// TIA Portal project "0000" (V15.1)

(* hardware
DEVICE "S7-1200-Station_1"  S7-1200 Station
   slot 0: "Baugruppenträger_0"  S7-1200 Rack  Rack  V1.0
   slot 1: "0000"  CPU 1214C DC/DC/DC  6ES7 214-1AG40-0XB0  V4.3
DEVICE "S7300/ET200M-Station_1"  S7-300 station
   slot 0: "Profilschiene_0"  Rail  6ES7 390-1***0-0AA0
   slot 2: "0001"  CPU 317-2 PN/DP  6ES7 317-2EK13-0AB0  V2.6
      slot 1: "MPI/DP-Schnittstelle_1"  X1
      slot 2: "PROFINET-Schnittstelle_1"  PN-IO
         slot 1: "Port_1"  Port
*)

// ===== PLC "0000"  CPU 1214C DC/DC/DC =====

VAR_GLOBAL   // PLC tag table "Standard-Variablentabelle"
   "Clock_Byte" AT %MB1 : Byte;
   "Clock_10Hz" AT %M1.0 : Bool;
   "Clock_5Hz" AT %M1.1 : Bool;
   "Clock_2.5Hz" AT %M1.2 : Bool;
   "Clock_2Hz" AT %M1.3 : Bool;
   "Clock_1.25Hz" AT %M1.4 : Bool;
   "Clock_1Hz" AT %M1.5 : Bool;
   "Clock_0.625Hz" AT %M1.6 : Bool;
   "Clock_0.5Hz" AT %M1.7 : Bool;
   "System_Byte" AT %MB0 : Byte;
   "FirstScan" AT %M0.0 : Bool;
   "DiagStatusUpdate" AT %M0.1 : Bool;
   "AlwaysTRUE" AT %M0.2 : Bool;
   "AlwaysFALSE" AT %M0.3 : Bool;
   "Enable_Communication" AT %M100.0 : Bool;
   "Save_Data" AT %M100.1 : Bool;
END_VAR

TYPE "_CSV_Data_UDT"
   STRUCT
      "example Bool" : Bool;   // this is a comment for Bool in UDT
   END_STRUCT;
END_TYPE

TYPE "_CSV_Data"
TITLE = has no title
// some comment
   STRUCT
      Save_Data : Bool := True;   // Trigger to save the data
      example_Byte : Byte := 16#2;   // this is a comment for example_Byte
      example_Word : Word := 16#FF;   // this is a comment for this is a comment for example_Word
      example_Dword : DWord := 16#FFFF;   // this is a comment for example_Dword
      example_Int : Int := 3;   // this is a comment for example_Int
      example_Dint : DInt := 5;   // this is a comment for example_Dint
      example_String : String := 'This is an example Text';   // this is a comment for example_String
      example_array : Array[0..5] of Bool;   // this is a comment for example_array
      example_UDT : "_CSV_Data_UDT";   // this is a comment for example UDT
   END_STRUCT;
END_TYPE

DATA_BLOCK "ConPlc_DB"   // DB1
{ S7_Optimized_Access := 'TRUE' }
VERSION : 0.1
// stored: InstanceOfName ConPlc
"ConPlc"
BEGIN
END_DATA_BLOCK

DATA_BLOCK "CSV"   // DB3
{ S7_Optimized_Access := 'FALSE' }
VERSION : 0.1
   VAR
      Data : "_CSV_Data";
   END_VAR
BEGIN
END_DATA_BLOCK

FUNCTION_BLOCK "ConPlc"   // FB1000, SCL
{ S7_Optimized_Access := 'TRUE' }
VERSION : 0.1
   VAR_INPUT
      ACTIVATE : Bool := False;   // activate connection
      TACT : Bool := False;   // tact
      CONN_ID : Conn_Ouc := 16#1;   // connection reference / identifier
      HW_ID : Hw_Any := 64;   // HW-identifier of IE-interface submodule
      CONN_Type : Byte := 16#0B;   // type of connection: 11=TCP/IP, 19=UDP (17=TCP/IP)
      IP_ADDR_1 : Byte := 16#C0;   // IPv4 address
      IP_ADDR_2 : Byte := 16#A8;   // IPv4 address
      IP_ADDR_3 : Byte := 16#00;   // IPv4 address
      IP_ADDR_4 : Byte := 16#1E;   // IPv4 address
      PORT_Remote : UInt := 2000;   // remote UDP/TCP port number
      PORT_Local : UInt := 2000;   // local UDP/TCP port number
   END_VAR
   VAR_OUTPUT
      Saved : Bool := False;   // CSV is saved
      Recieved : Bool := False;   // Data is recieved
   END_VAR
   VAR_IN_OUT
      DATA : Variant;
   END_VAR
   VAR
      ACT_CONN : Bool;
      CONN_ESTABLISHED : Bool;
      DONE_CONN : Bool;
      BUSY_CONN : Bool;
      ERROR_CONN : Bool;
      STATUS_CONN : Word;
      DONE_SEND : Bool;
      BUSY_SEND : Bool;
      ERROR_SEND : Bool;
      STATUS_SEND : Word;
      ACT_SEND : Bool;
      NDR_RECV : Bool;
      BUSY_RECV : Bool;
      ERROR_RECV : Bool;
      STATUS_RECV : Word;
      RCVD_LEN : UDInt;
      ACT_RECV : Bool;
      DONE_DISCON : Bool;
      BUSY_DISCON : Bool;
      ERROR_DISCON : Bool;
      STATUS_DISCON : Word;
      ACT_DISCON : Bool;
      TRIGGER : Bool;
      TRIGGER_MEM : Bool;
      RECV : Array[0..9] of Char;
      TCON_IDB : TCON;
      TSEND_IDB : TSEND;
      TRCV_IDB : TRCV;
      TDISCON_IDB : TDISCON;
      CONN_PARAMETER : TCON_IP_v4;
      TON_RESET : TON_TIME;
   END_VAR
   VAR_TEMP
      recv_str : String[10];
   END_VAR
   // CONN_PARAMETER.InterfaceId := 64;
   // CONN_PARAMETER.ID := 16#1;
   // CONN_PARAMETER.ConnectionType := 16#0B;
   // CONN_PARAMETER.ActiveEstablished := False;
   // CONN_PARAMETER.RemoteAddress.ADDR[1] := 16#C0;
   // CONN_PARAMETER.RemoteAddress.ADDR[2] := 16#A8;
   // CONN_PARAMETER.RemoteAddress.ADDR[3] := 16#00;
   // CONN_PARAMETER.RemoteAddress.ADDR[4] := 16#1E;
   // CONN_PARAMETER.RemotePort := 2000;
   // CONN_PARAMETER.LocalPort := 2000;
BEGIN
   REGION set connection data
       #CONN_PARAMETER.ID := #CONN_ID;
       #CONN_PARAMETER.InterfaceId := #HW_ID;
       #CONN_PARAMETER.ActiveEstablished := TRUE;
       #CONN_PARAMETER.ConnectionType := #CONN_Type;
       #CONN_PARAMETER.RemoteAddress.ADDR[1] := #IP_ADDR_1;
       #CONN_PARAMETER.RemoteAddress.ADDR[2] := #IP_ADDR_2;
       #CONN_PARAMETER.RemoteAddress.ADDR[3] := #IP_ADDR_3;
       #CONN_PARAMETER.RemoteAddress.ADDR[4] := #IP_ADDR_4;
       #CONN_PARAMETER.RemotePort := #PORT_Remote;
       #CONN_PARAMETER.LocalPort := #PORT_Local;
   END_REGION

   REGION create trigger
       #TRIGGER := #TACT AND NOT #TRIGGER_MEM;
       #TRIGGER_MEM := #TACT;
   END_REGION

   REGION connect
       //connect enable
       IF #ACTIVATE AND NOT #CONN_ESTABLISHED THEN
           #ACT_CONN := True;
       END_IF;
       //connect
       #TCON_IDB(REQ       := #ACT_CONN AND #TRIGGER,
                 ID        := #CONN_ID,
                 DONE      => #DONE_CONN,
                 BUSY      => #BUSY_CONN,
                 ERROR     => #ERROR_CONN,
                 STATUS    => #STATUS_CONN,
                 CONNECT   := #CONN_PARAMETER);
       //connect done
       IF #DONE_CONN THEN
           #CONN_ESTABLISHED := True;
           #ACT_CONN := False;
       END_IF;
   END_REGION

   REGION send
       //send enable
       #ACT_SEND := #CONN_ESTABLISHED AND #TRIGGER AND NOT #BUSY_SEND;
       //send
       #TSEND_IDB(REQ      := #ACT_SEND,
                  ID       := #CONN_ID,
                  LEN      := 0,
                  DONE     => #DONE_SEND,
                  BUSY     => #BUSY_SEND,
                  ERROR    => #ERROR_SEND,
                  STATUS   => #STATUS_SEND,
                  DATA     := #DATA);
   END_REGION

   REGION recieve

       //revieve enable
       #ACT_RECV := #CONN_ESTABLISHED;
       //recieve
       #TRCV_IDB(EN_R      := #ACT_RECV,
                 ID        := #CONN_ID,
                 LEN       := 10,
                 ADHOC     := TRUE,
                 NDR       => #NDR_RECV,
                 BUSY      => #BUSY_RECV,
                 ERROR     => #ERROR_RECV,
                 STATUS    => #STATUS_RECV,
                 RCVD_LEN  => #RCVD_LEN,
                 DATA      := #RECV);

       //put recieved Bytes in String
       Chars_TO_Strg(Chars:=#RECV, pChars:=0, Cnt:=10, Strg=>#recv_str);

       //check recieved data
       #Saved := #NDR_RECV AND (#recv_str = 'Saved     ');
       #Recieved := #NDR_RECV AND (#recv_str = 'Recieved  ');

   END_REGION

   REGION disconnect
       //disconnect enable
       #TON_RESET(IN := #ACTIVATE AND NOT #CONN_ESTABLISHED,
                  PT := T#5s);
       #ACT_DISCON := (#TON_RESET.Q) OR (NOT #ACTIVATE);
       //disconnect
       #TDISCON_IDB(REQ    := #ACT_DISCON,
                    ID     := #CONN_ID,
                    DONE   => #DONE_DISCON,
                    BUSY   => #BUSY_DISCON,
                    ERROR  => #ERROR_DISCON,
                    STATUS => #STATUS_DISCON);

       //disconnect done
       IF NOT #ACTIVATE THEN
           #CONN_ESTABLISHED := False;
           #ACT_CONN := False;
       END_IF;
   END_REGION
END_FUNCTION_BLOCK

ORGANIZATION_BLOCK "Main"   // OB1, FBD, ProgramCycle
TITLE = "Main Program Sweep (Cycle)"
{ S7_Optimized_Access := 'TRUE' }
VERSION : 0.1
   VAR_INPUT
      Initial_Call : Bool;   // Initial call of this OB
      Remanence : Bool;   // =True, if remanent data are available
   END_VAR
   VAR_TEMP
      retval : Int;
      saved : Bool;
      recieved : Bool;
   END_VAR
BEGIN

REGION Network 1: Collect Data
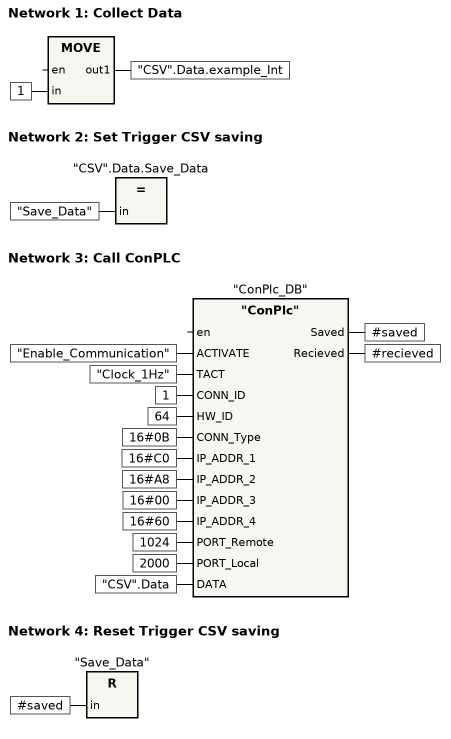
   "CSV".Data.example_Int := 1;
END_REGION

REGION Network 2: Set Trigger CSV saving
   "CSV".Data.Save_Data := "Save_Data";
END_REGION

REGION Network 3: Call ConPLC
   "ConPlc_DB"(ACTIVATE := "Enable_Communication",   // "ConPlc"
               TACT := "Clock_1Hz",
               CONN_ID := 1,
               HW_ID := 64,
               CONN_Type := 16#0B,
               IP_ADDR_1 := 16#C0,
               IP_ADDR_2 := 16#A8,
               IP_ADDR_3 := 16#00,
               IP_ADDR_4 := 16#60,
               PORT_Remote := 1024,
               PORT_Local := 2000,
               DATA := "CSV".Data,
               Saved => #saved,
               Recieved => #recieved);
END_REGION

REGION Network 4: Reset Trigger CSV saving
   IF #saved THEN "Save_Data" := FALSE; END_IF;
END_REGION
END_ORGANIZATION_BLOCK

// ===== PLC "0001"  CPU 317-2 PN/DP =====

VAR_GLOBAL   // PLC tag table "Standard-Variablentabelle"
   "Clock_Byte" AT %MB1 : Byte;
   "Clock_10Hz" AT %M1.0 : Bool;
   "Clock_5Hz" AT %M1.1 : Bool;
   "Clock_2.5Hz" AT %M1.2 : Bool;
   "Clock_2Hz" AT %M1.3 : Bool;
   "Clock_1.25Hz" AT %M1.4 : Bool;
   "Clock_1Hz" AT %M1.5 : Bool;
   "Clock_0.625Hz" AT %M1.6 : Bool;
   "Clock_0.5Hz" AT %M1.7 : Bool;
   "Enable_Communication" AT %M100.0 : Bool;
   "Save_Data" AT %M100.1 : Bool;
END_VAR

TYPE "_CSV_Data_UDT"
   STRUCT
      "example Bool" : Bool;   // this is a comment for Bool in UDT
   END_STRUCT;
END_TYPE

TYPE "_CSV_Data"
TITLE = has no title
// some comment
   STRUCT
      Save_Data : Bool := True;   // Trigger to save the data
      example_Byte : Byte := 16#2;   // this is a comment for example_Byte
      example_Word : Word := 16#FF;   // this is a comment for this is a comment for example_Word
      example_Dword : DWord := 16#FFFF;   // this is a comment for example_Dword
      example_Int : Int := 3;   // this is a comment for example_Int
      example_Dint : DInt := 5;   // this is a comment for example_Dint
      example_String : String := 'This is an example Text';   // this is a comment for example_String
      example_array : Array[0..5] of Bool;   // this is a comment for example_array
      example_UDT : "_CSV_Data_UDT";   // this is a comment for example UDT
   END_STRUCT;
END_TYPE

DATA_BLOCK "ConPlc_DB"   // DB1
{ S7_Optimized_Access := 'FALSE' }
VERSION : 0.1
// stored: InstanceOfName ConPlc
"ConPlc"
BEGIN
   ACTIVATE := TRUE;
   TACT := TRUE;
   CONN_ID := 16#0001;
   Saved := FALSE;
   Recieved := FALSE;
   DATA := P#DB3.DBX0.0 BYTE 274;
   ACT_CONN := TRUE;
   STATUS_CONN := 16#7000;
   STATUS_SEND := 16#7000;
   STATUS_RECV := 16#7000;
   STATUS_DISCON := 16#7000;
   ACT_DISCON := TRUE;
   TRIGGER := TRUE;
   TRIGGER_MEM := TRUE;
   RECV[0] := ' ';
   RECV[1] := ' ';
   RECV[2] := ' ';
   RECV[3] := ' ';
   RECV[4] := ' ';
   RECV[5] := ' ';
   RECV[6] := ' ';
   RECV[7] := ' ';
   RECV[8] := ' ';
   RECV[9] := ' ';
   TCON_IDB.REQ := TRUE;
   TCON_IDB.ID := 16#0001;
   TCON_IDB.STATUS := 16#7000;
   TCON_IDB.CONNECT := P#DB1.DBX122.0 BYTE 64;
   TSEND_IDB.ID := 16#0001;
   TSEND_IDB.STATUS := 16#7000;
   TSEND_IDB.DATA := P#DB3.DBX0.0 BYTE 274;
   TRCV_IDB.ID := 16#0001;
   TRCV_IDB.LEN := 10;
   TRCV_IDB.STATUS := 16#7000;
   TRCV_IDB.DATA := P#DB1.DBX36.0 CHAR 10;
   TDISCON_IDB.REQ := TRUE;
   TDISCON_IDB.ID := 16#0001;
   TDISCON_IDB.STATUS := 16#7000;
   TON_RESET.IN := TRUE;
   TON_RESET.PT := T#5S;
   TON_RESET.Q := TRUE;
   TON_RESET.ET := T#5S;
END_DATA_BLOCK

DATA_BLOCK "CSV"   // DB3
{ S7_Optimized_Access := 'FALSE' }
VERSION : 0.1
   VAR
      Data : "_CSV_Data";
   END_VAR
BEGIN
END_DATA_BLOCK

FUNCTION_BLOCK "ConPlc"   // FB1000, SCL
{ S7_Optimized_Access := 'FALSE' }
VERSION : 0.1
   VAR_INPUT
      ACTIVATE : Bool := False;   // activate connection
      TACT : Bool := False;   // tact
      CONN_ID : Word := 16#1;   // connection reference / identifier
   END_VAR
   VAR_OUTPUT
      Saved : Bool := False;   // CSV is saved
      Recieved : Bool := False;   // Data is recieved
   END_VAR
   VAR_IN_OUT
      DATA : ANY;
   END_VAR
   VAR
      ACT_CONN : Bool;
      CONN_ESTABLISHED : Bool;
      DONE_CONN : Bool;
      BUSY_CONN : Bool;
      ERROR_CONN : Bool;
      STATUS_CONN : Word;
      DONE_SEND : Bool;
      BUSY_SEND : Bool;
      ERROR_SEND : Bool;
      STATUS_SEND : Word;
      ACT_SEND : Bool;
      NDR_RECV : Bool;
      BUSY_RECV : Bool;
      ERROR_RECV : Bool;
      STATUS_RECV : Word;
      RCVD_LEN : Int;
      ACT_RECV : Bool;
      DONE_DISCON : Bool;
      BUSY_DISCON : Bool;
      ERROR_DISCON : Bool;
      STATUS_DISCON : Word;
      ACT_DISCON : Bool;
      TRIGGER : Bool;
      TRIGGER_MEM : Bool;
      RECV : Array[0..9] of Char;
      TCON_IDB : TCON;
      TSEND_IDB : TSEND;
      TRCV_IDB : TRCV;
      TDISCON_IDB : TDISCON;
      CONN_PARAMETER : TCON_PAR;
      TON_RESET : TON;
   END_VAR
   VAR_TEMP
      recv_str : String[10];
      cnt : Int;
      retval : Int;
   END_VAR
BEGIN
   REGION create trigger
       #TRIGGER := #TACT AND NOT #TRIGGER_MEM;
       #TRIGGER_MEM := #TACT;
   END_REGION

   REGION connect
       //connect enable
       IF #ACTIVATE AND NOT #CONN_ESTABLISHED THEN
           #ACT_CONN := True;
       END_IF;

       //connect
       #TCON_IDB(REQ       := #ACT_CONN AND #TRIGGER,
                 ID        := #CONN_ID,
                 DONE      => #DONE_CONN,
                 BUSY      => #BUSY_CONN,
                 ERROR     => #ERROR_CONN,
                 STATUS    => #STATUS_CONN,
                 CONNECT   := #CONN_PARAMETER);
       //connect done
       IF #DONE_CONN THEN
           #CONN_ESTABLISHED := True;
           #ACT_CONN := False;
       END_IF;
   END_REGION

   REGION send
       //send enable
       #ACT_SEND := #CONN_ESTABLISHED AND #TRIGGER AND NOT #BUSY_SEND;
       //send
       #TSEND_IDB(REQ      := #ACT_SEND,
                  ID       := #CONN_ID,
                  LEN      := 0,
                  DONE     => #DONE_SEND,
                  BUSY     => #BUSY_SEND,
                  ERROR    => #ERROR_SEND,
                  STATUS   => #STATUS_SEND,
                  DATA     := #DATA);
   END_REGION

   REGION recieve

       //revieve enable
       #ACT_RECV := #CONN_ESTABLISHED;
       //recieve
       #TRCV_IDB(EN_R      := #ACT_RECV,
                 ID        := #CONN_ID,
                 LEN       := 10,
                 NDR       => #NDR_RECV,
                 BUSY      => #BUSY_RECV,
                 ERROR     => #ERROR_RECV,
                 STATUS    => #STATUS_RECV,
                 RCVD_LEN  => #RCVD_LEN,
                 DATA      := #RECV);

       //put recieved Bytes in String
       #retval := BLKMOV(SRCBLK:=#RECV, DSTBLK=>#recv_str);

       //check recieved data
       #Saved := #NDR_RECV AND (#recv_str S_COMP 'Saved     ');
       #Recieved := #NDR_RECV AND (#recv_str S_COMP 'Recieved  ');

   END_REGION

   REGION disconnect
       //disconnect enable
       #TON_RESET(IN := #ACTIVATE AND NOT #CONN_ESTABLISHED,
                  PT := T#5s);
       #ACT_DISCON := (#TON_RESET.Q) OR (NOT #ACTIVATE);
       //disconnect
       #TDISCON_IDB(REQ    := #ACT_DISCON,
                    ID     := #CONN_ID,
                    DONE   => #DONE_DISCON,
                    BUSY   => #BUSY_DISCON,
                    ERROR  => #ERROR_DISCON,
                    STATUS => #STATUS_DISCON);

       //disconnect done
       IF NOT #ACTIVATE THEN
           #CONN_ESTABLISHED := False;
           #ACT_CONN := False;
       END_IF;
   END_REGION
END_FUNCTION_BLOCK

ORGANIZATION_BLOCK "Main"   // OB1, FBD
TITLE = "Main Program Sweep (Cycle)"
{ S7_Optimized_Access := 'FALSE' }
VERSION : 0.1
   VAR_TEMP
      OB1_EV_CLASS : Byte;   // Bits 0-3 = 1 (Coming event), Bits 4-7 = 1 (Event class 1)
      OB1_SCAN_1 : Byte;   // 1 (Cold restart scan 1 of OB 1), 3 (Scan 2-n of OB 1)
      OB1_PRIORITY : Byte;   // Priority of OB Execution
      OB1_OB_NUMBR : Byte;   // 1 (Organization block 1, OB1)
      OB1_RESERVED_1 : Byte;   // Reserved for system
      OB1_RESERVED_2 : Byte;   // Reserved for system
      OB1_PREV_CYCLE : Int;   // Cycle time of previous OB1 scan (milliseconds)
      OB1_MIN_CYCLE : Int;   // Minimum cycle time of OB1 (milliseconds)
      OB1_MAX_CYCLE : Int;   // Maximum cycle time of OB1 (milliseconds)
      OB1_DATE_TIME : Date_And_Time;   // Date and time OB1 started
      saved : Bool;
      recieved : Bool;
   END_VAR
BEGIN

REGION Network 1: Collect Data
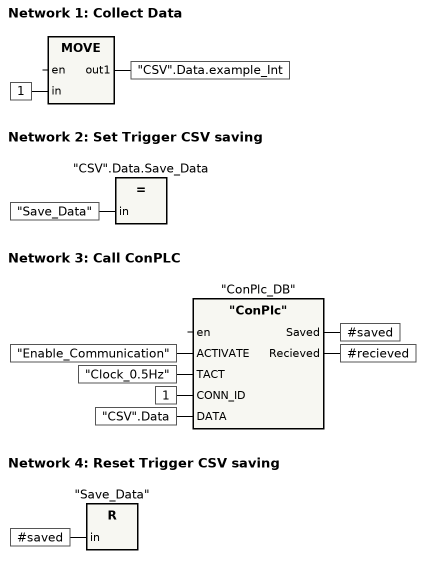
   "CSV".Data.example_Int := 1;
END_REGION

REGION Network 2: Set Trigger CSV saving
   "CSV".Data.Save_Data := "Save_Data";
END_REGION

REGION Network 3: Call ConPLC
   "ConPlc_DB"(ACTIVATE := "Enable_Communication",   // "ConPlc"
               TACT := "Clock_0.5Hz",
               CONN_ID := 1,
               DATA := "CSV".Data,
               Saved => #saved,
               Recieved => #recieved);
END_REGION

REGION Network 4: Reset Trigger CSV saving
   IF #saved THEN "Save_Data" := FALSE; END_IF;
END_REGION
END_ORGANIZATION_BLOCK